(* IEC 61131-3 sources: our-getting-started/src, 8 files *)

(* ---- OperatingMode.st ---- *)
NAMESPACE Siemens.Ax
    /// An enumeration with the values 'Automatic', 'Manual', 'Maintenance' where
    /// the default value is 'Manual'
    TYPE
        OperatingMode : (Automatic, Manual, Maintenance) := Manual;
    END_TYPE
END_NAMESPACE

(* ---- IOperatingModeController.st ---- *)
NAMESPACE Siemens.Ax

    /// Interface for OperatingModeController
    INTERFACE IOperatingModeController
        METHOD SetOperatingMode
            VAR_INPUT
                mode : OperatingMode;
            END_VAR
        END_METHOD
        METHOD GetOperatingMode : OperatingMode
        END_METHOD
    END_INTERFACE

END_NAMESPACE

(* ---- Add.st ---- *)
// Functions including overloading of functions

NAMESPACE Siemens.Ax
    /// Returns the sum of i1 + i2 ot type INT
    FUNCTION Add : DINT
        VAR_INPUT
            i1 : INT;
            i2 : INT;
        END_VAR
            Add := TO_DINT(i1) + TO_DINT(i2);
            // To force an error in AxUnit, uncomment the following line
            // Add := i1 + i2; // 32000 + 32000 leads to an integer overflow
    END_FUNCTION

    /// Returns the sum of i1 + i2 ot type LREAL
    FUNCTION Add : LREAL
        VAR_INPUT
            i1 : LREAL;
            i2 : LREAL;
        END_VAR
        VAR_TEMP
            lb, ub, i : DINT;
        END_VAR

        FOR i := lb TO ub DO
            ;
        END_FOR;
    END_FUNCTION

END_NAMESPACE

(* ---- HelloWorldFunction.st ---- *)
NAMESPACE Siemens.Ax
    /// Returns the value 'Hello AX World'
    FUNCTION HelloWorldFunction : STRING
        HelloWorldFunction := 'Hello AX World';
    END_FUNCTION
END_NAMESPACE

(* ---- OperatingModeController.st ---- *)
NAMESPACE Siemens.Ax

    /// OperatingModeController is an example for using OOP features in ST
    /// In this example you can:
    /// Set the operatinfg mode with SetOperatingMode(mode := [Automatic, Manual, Maintenance])
    /// Read the active operating mode with GetOperatingMode()
    /// Note: This is just an example without any productive character
    CLASS OperatingModeController
        IMPLEMENTS IOperatingModeController
        VAR PUBLIC
            Zone : INT;
        END_VAR
        VAR PROTECTED
            _operatingMode : OperatingMode;
        END_VAR
        /// Set the active operating mode
        METHOD PUBLIC SetOperatingMode
            VAR_INPUT
                mode : OperatingMode;
            END_VAR
            _operatingMode := mode;
        END_METHOD
        /// Returns the active operating mode
        METHOD PUBLIC GetOperatingMode : OperatingMode
            GetOperatingMode := _operatingMode;
        END_METHOD
    END_CLASS

END_NAMESPACE

(* ---- OperatingModeControllerExt.st ---- *)
NAMESPACE Siemens.Ax

    /// In this example, the standard OperatingModeController will be extendet by
    /// the method GetZoneStatusAsInt(). This coud be an extension to assign a
    /// the status to an HMI where a INT value is requiired
    CLASS OperatingModeControllerExt EXTENDS OperatingModeController

        METHOD PUBLIC GetZoneStatusAsInt : INT
            // calling a private method with THIS-Operator
            GetZoneStatusAsInt := THIS.CalculateZoneStatus(_operatingMode);
        END_METHOD
        /// Calculate the ZoneNumber depending on active operating mode and zone number
        METHOD PRIVATE CalculateZoneStatus : INT
            VAR_INPUT
                mode : OperatingMode;
            END_VAR
            CASE mode OF
                OperatingMode#Manual:
                    CalculateZoneStatus := Zone;
                    RETURN;
                OperatingMode#Automatic:
                    CalculateZoneStatus := Zone * 10;
                    RETURN;
                OperatingMode#Maintenance:
                    CalculateZoneStatus := 0;
                    RETURN;
            END_CASE;
        END_METHOD
    END_CLASS

END_NAMESPACE

(* ---- configuration.st ---- *)
USING Siemens.Ax;

CONFIGURATION MyConfiguration
    // Create main task
    TASK Main (PRIORITY := 1);
    // Assign MyProgram to main (cyclic) task
    PROGRAM P1 WITH Main: MyProgram;
    VAR_GLOBAL
        v1 : INT := 4; // initial values
        v2 : INT;
        sum : DINT;
        myString : STRING := 'Hello World';
        // OperatingModes with initializer for VAR_PUBLICs
        OpModeZone1 : OperatingModeController := (Zone := 1);
        OpModeZone2 : OperatingModeController := (Zone := 2);
    END_VAR
END_CONFIGURATION

(* ---- program.st ---- *)
USING Siemens.Ax;
PROGRAM MyProgram
    VAR_EXTERNAL
        myString : String;
        v1 : INT;
        v2 : INT;
        sum : DINT;

        // OperatingModes with initializer for VAR_PUBLICs
        OpModeZone1 : OperatingModeController;
        OpModeZone2 : OperatingModeController;

    END_VAR

    VAR

    END_VAR

    VAR_TEMP

    END_VAR

    // Call function Add(i1, i2);
    sum := Add(v1, v2);

    // Call function hello world fully qualified
    myString := Siemens.Ax.HelloWorldFunction();

END_PROGRAM
